PROGRAM MAIN
VAR
	a,b,c,d:int;
END_VAR

c:=a+b;

END_PROGRAM

(* stored: Version 1.1.0.1, ProductVersion 3.1.4024.3
   POU MAIN: Id {b98af3ec-355a-4bfd-b73e-6129ab2fe437}, SpecialFunc None *)
